//-----------------------------------------------------------------------------------------
//
//                  				ST_HMI_Doors
//
//								Structure portes HMI			
//-----------------------------------------------------------------------------------------
//
//Auteur: G.GOETZ
//Création: 20.02.2026
//Dernière modification : 20.02.2026 (G.GOETZ)
//       			
//-----------------------------------------------------------------------------------------
//
//     							Liste des modifications  	
//
// 20.02.2026 (G.GOETZ) -> Création		
//-----------------------------------------------------------------------------------------

TYPE ST_HMI_Doors :
STRUCT

	(** SETUP FLAG **)
		bDoorUnlockForce : BOOL ; // Door unlocking force

END_STRUCT
END_TYPE

(* stored: Version 1.1.0.1, ProductVersion 3.1.4026.17
   DUT ST_HMI_Doors: Id {639b00cc-bc27-4b90-a6aa-9e14b8039040} *)
